LAYER Nereda
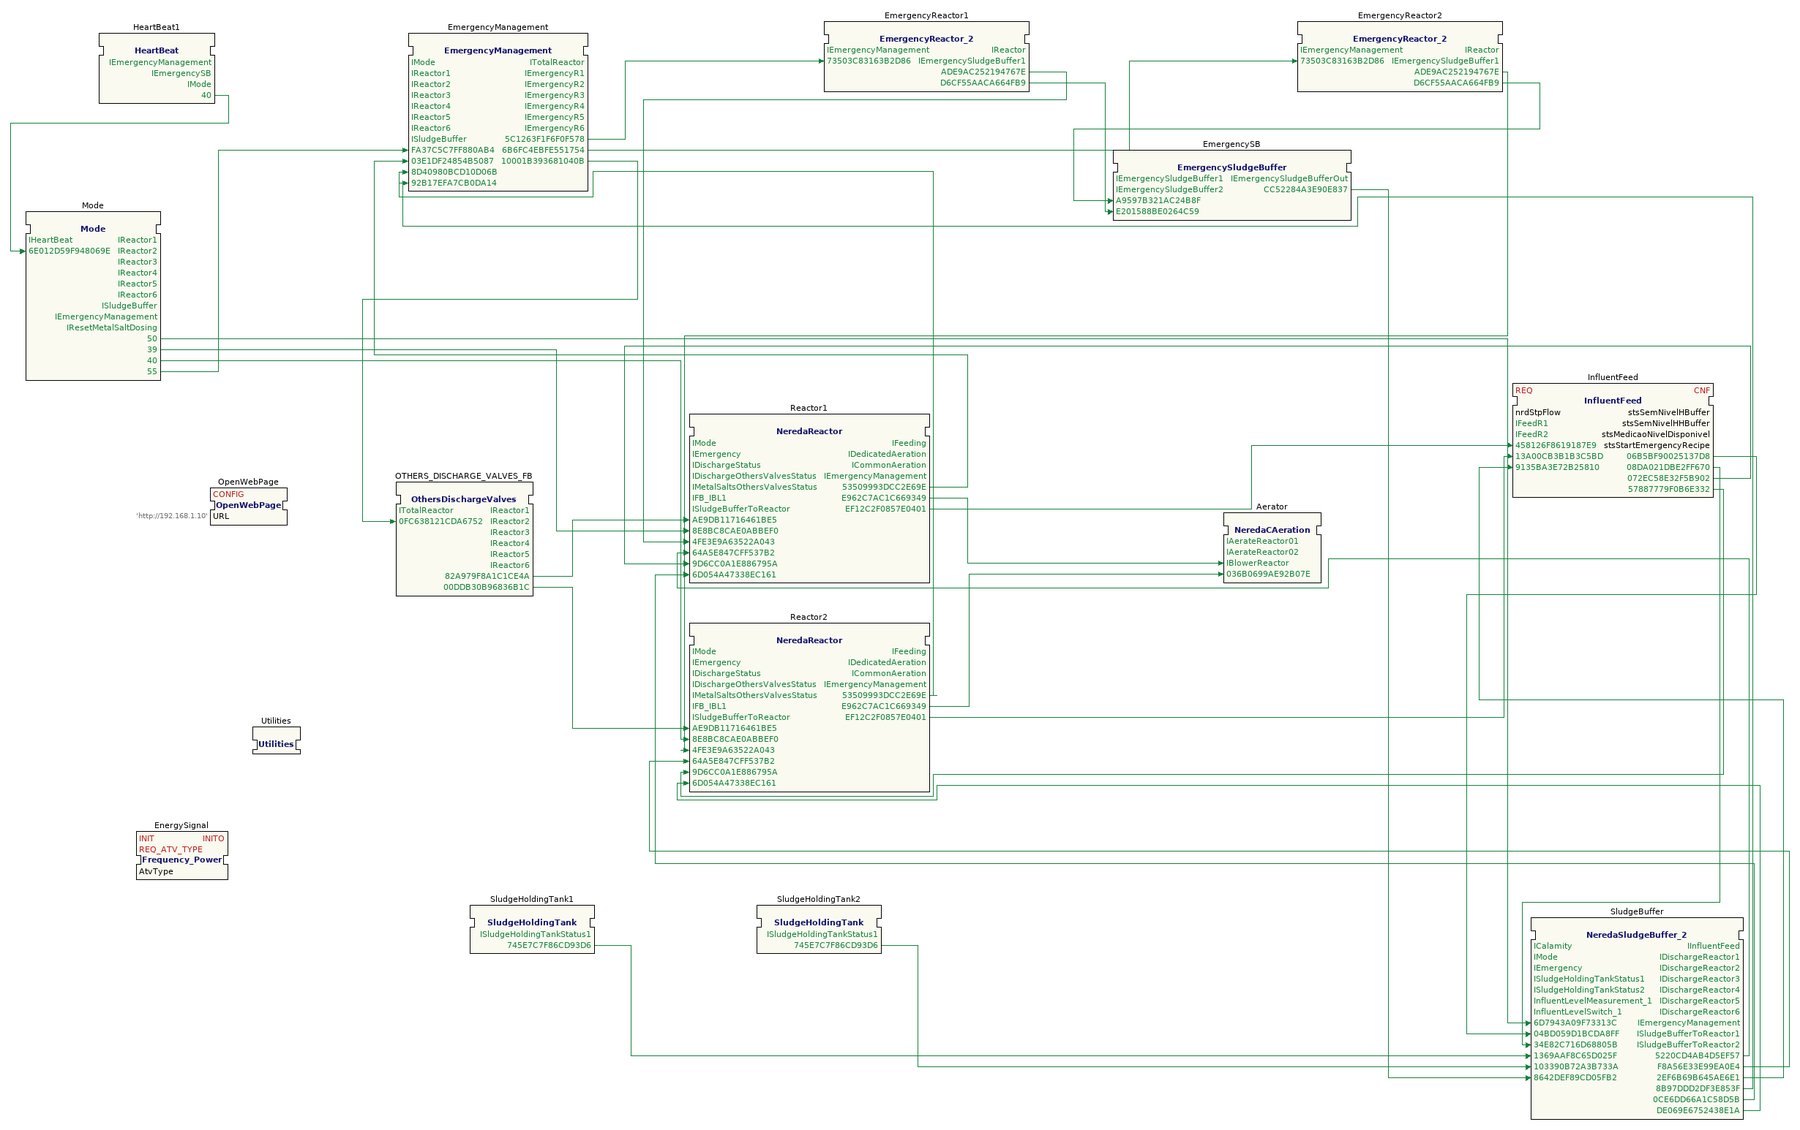
  (* NEREDA REACTORS *)
  (* NEREDA PROCESS - HIDRYCO *)
  (* EMERGENCY RECIPIE *)
  (* NEREDA EQUIPMENT *)
  (* NEREDA AERATION *)
  (* INFLUENT FEED *)
  (* EFFLUENT *)
  (* SLUDGE BUFFER *)
  (* METAL SALT DOSING *)
  (* SLUDGE HOLDING TANK *)
  FBS
    Mode : Mode; {SET_ATTRIBUTE(CompilerOptions, CheckConnectionsStrictly=False)}
    OpenWebPage : OpenWebPage(URL := 'http://192.168.1.10');
    OTHERS_DISCHARGE_VALVES_FB : OthersDischargeValves;
    EmergencyManagement : EmergencyManagement;
    Utilities : Utilities;
    EnergySignal : Frequency_Power;
    HeartBeat1 : HeartBeat;
    Aerator : NeredaCAeration;
    SludgeBuffer : NeredaSludgeBuffer_2;
    SludgeHoldingTank1 : SludgeHoldingTank;
    SludgeHoldingTank2 : SludgeHoldingTank;
    Reactor1 : NeredaReactor;
    Reactor2 : NeredaReactor;
    EmergencySB : EmergencySludgeBuffer;
    EmergencyReactor1 : EmergencyReactor_2;
    EmergencyReactor2 : EmergencyReactor_2;
    InfluentFeed : InfluentFeed;
  END_FBS
  ADAPTER_CONNECTIONS
    HeartBeat1.40 TO Mode.6E012D59F948069E;
    Mode.50 TO SludgeBuffer.6D7943A09F73313C;
    InfluentFeed.06B5BF90025137D8 TO SludgeBuffer.04BD059D1BCDA8FF;
    InfluentFeed.08DA021DBE2FF670 TO SludgeBuffer.34E82C716D68805B;
    SludgeHoldingTank1.745E7C7F86CD93D6 TO SludgeBuffer.1369AAF8C65D025F;
    SludgeHoldingTank2.745E7C7F86CD93D6 TO SludgeBuffer.103390B72A3B733A;
    OTHERS_DISCHARGE_VALVES_FB.82A979F8A1C1CE4A TO Reactor1.AE9DB11716461BE5;
    OTHERS_DISCHARGE_VALVES_FB.00DDB30B96836B1C TO Reactor2.AE9DB11716461BE5;
    Mode.39 TO Reactor1.8E8BC8CAE0ABBEF0;
    Mode.40 TO Reactor2.8E8BC8CAE0ABBEF0;
    Mode.55 TO EmergencyManagement.FA37C5C7FF880AB4;
    Reactor1.53509993DCC2E69E TO EmergencyManagement.03E1DF24854B5087;
    Reactor2.53509993DCC2E69E TO EmergencyManagement.8D40980BCD10D06B;
    EmergencyManagement.5C1263F1F6F0F578 TO EmergencyReactor1.73503C83163B2D86;
    EmergencyManagement.6B6FC4EBFE551754 TO EmergencyReactor2.73503C83163B2D86;
    Reactor1.E962C7AC1C669349 TO Aerator.IBlowerReactor;
    Reactor2.E962C7AC1C669349 TO Aerator.036B0699AE92B07E;
    Reactor1.EF12C2F0857E0401 TO InfluentFeed.458126F8619187E9;
    Reactor2.EF12C2F0857E0401 TO InfluentFeed.13A00CB3B1B3C5BD;
    EmergencyReactor1.ADE9AC252194767E TO Reactor1.4FE3E9A63522A043;
    EmergencyReactor2.ADE9AC252194767E TO Reactor2.4FE3E9A63522A043;
    SludgeBuffer.5220CD4AB4D5EF57 TO Reactor1.64A5E847CFF537B2;
    SludgeBuffer.F8A56E33E99EA0E4 TO Reactor2.64A5E847CFF537B2;
    SludgeBuffer.2EF6B69B645AE6E1 TO InfluentFeed.9135BA3E72B25810;
    EmergencyManagement.10001B393681040B TO OTHERS_DISCHARGE_VALVES_FB.0FC638121CDA6752;
    SludgeBuffer.8B97DDD2DF3E853F TO EmergencyManagement.92B17EFA7CB0DA14;
    EmergencyReactor2.D6CF55AACA664FB9 TO EmergencySB.A9597B321AC24B8F;
    EmergencyReactor1.D6CF55AACA664FB9 TO EmergencySB.E201588BE0264C59;
    InfluentFeed.072EC58E32F5B902 TO Reactor1.9D6CC0A1E886795A;
    InfluentFeed.57887779F0B6E332 TO Reactor2.9D6CC0A1E886795A;
    SludgeBuffer.0CE6DD66A1C58D5B TO Reactor1.6D054A47338EC161;
    SludgeBuffer.DE069E6752438E1A TO Reactor2.6D054A47338EC161;
    EmergencySB.CC52284A3E90E837 TO SludgeBuffer.8642DEF89CD05FB2;
  END_CONNECTIONS
END_LAYER
